INTERFACE I_coupler_execution

METHOD run : BOOL
VAR_INPUT
	sync_unit_ok : BOOL;
END_VAR
END_METHOD

END_INTERFACE

(* stored: Version 1.1.0.1, ProductVersion 3.1.4024.6
   Itf I_coupler_execution: Id {58bf683b-17fa-0ab4-29c4-de9a18a652f6}
   Method run: Id {141afd9f-2786-0c5e-00da-c6ddc0438cd2} *)
